(*			
	RafalOS
	Rafał Osajda		12.11.2025		TC 4024.66
	interfejs do przekazywania przy tworzeniu elementów
*)
INTERFACE ITF_HMIEMenu_HMI_Init EXTENDS ITF_BaseControlElement, ITF_HMIEMenu_HMI_Connector

END_INTERFACE

(* stored: Version 1.1.0.1
   Itf ITF_HMIEMenu_HMI_Init: Id {3d5bacc6-1c37-046a-128d-335ccf25c56b} *)
